TYPE DUT_StaHistory :
STRUCT
		History:ARRAY [1..500] OF STRING[100];
END_STRUCT
END_TYPE

(* stored: Version 1.1.0.1, ProductVersion 3.1.4024.9
   DUT DUT_StaHistory: Id {d02c2898-9095-4bfa-9d63-0bc815c3ee2f} *)
